FUNCTION_BLOCK FB_PB_TransportControlEmulation EXTENDS FB_TransportControlEmulation
(**************************************************************************************
 * 	Application		:	Pro Box
 *	Revision		:	$Revision:  $
 *	Revision date	:	$Date: $
 *	Last changed by	:	$Author: q8hedls $
 *	URL				:	$$
 *
 *	Purpose			:	Override BCF Transport control emulation
 *
 * ------------------------------------------------------------------------------------
 *	Copyright Swisslog [IP AG], Switzerland. All rights reserved.
 * 
 * ------------------------------------------------------------------------------------
 *	
 **************************************************************************************)
VAR_INPUT
	
END_VAR

VAR_IN_OUT
	//ZoneData				: ST_ZoneDataEmulation; // Zone data
END_VAR


SUPER^(ZoneData :=ZoneData);

END_FUNCTION_BLOCK

(* stored: Version 1.1.0.1, ProductVersion 3.1.4024.4
   POU FB_PB_TransportControlEmulation: Id {b44972de-ebb2-4321-a955-69dc6ed1b94f}, SpecialFunc None *)
